FUNCTION_BLOCK PAEActValve2_1plus2 EXTENDS PAEActuator2way_1plus2
VAR_INPUT
END_VAR
VAR_OUTPUT
END_VAR
VAR
END_VAR

END_FUNCTION_BLOCK

(* stored: Version 1.1.0.1, ProductVersion 3.1.4020.12
   POU PAEActValve2_1plus2: Id {6de9fff4-e55b-4a36-9dac-bd7d8de4a28d}, SpecialFunc None *)
